// TIA Portal V16 export
// export: Created 2021-04-06T19:52:16.9011384Z, ExportSetting WithDefaults, DisplayName Totally Integrated Automation Portal, DisplayVersion V16, DisplayName TIA Portal Version Control Interface, DisplayVersion V16, DisplayName TIA Portal Openness, DisplayVersion V16, DisplayName STEP 7 Professional, DisplayVersion V16, DisplayName STEP 7 Safety, DisplayVersion V16, DisplayName WinCC Unified SCADA Engineering System, DisplayVersion V16
FUNCTION_BLOCK "workInConveyer_AM"   // FB6, LAD
{ S7_Optimized_Access := 'TRUE' }
VERSION : 0.1
// stored: AutoNumber true, IsIECCheckEnabled false, IsRetainMemResEnabled false, MemoryReserve 100, SetENOAutomatically false, UDAEnableTagReadback false
   VAR_INPUT
      enableWork : Bool;   // разрешение работы
      "setSpeed%Int" : Int;   // уставка скорости
      sensorOverflow : Bool;   // датчик пересыпа
   END_VAR
   VAR_OUTPUT
      startinConveyor : Bool;   // запуск конвейера
      "setSpeed%Real" : Real;
   END_VAR
   VAR
      tonOverflowTable : TON_TIME;   // задержка на включение сигнала пересыпа
      tofOverflowTable : TOF_TIME;   // задержка на выключение сигнала пересыпа
      isOverFlowTable : Bool;   // сигнал сработки сигнала пересыпа
   END_VAR
BEGIN

REGION Network 1: сигнал сработки сигнала пересыпа
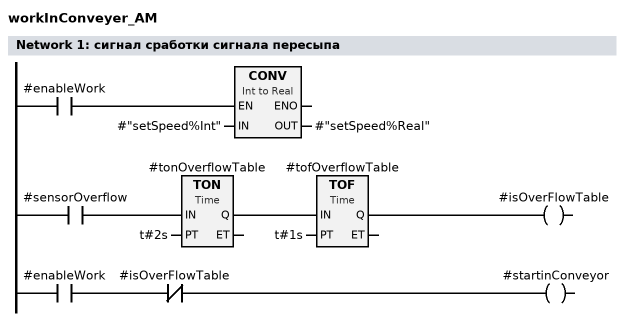
   RUNG wire#powerrail
      Contact( #enableWork )
      { S7_Templates := "[SrcType := Int, DestType := Real]" } Convert(in := #"setSpeed%Int", out => #"setSpeed%Real")
   END_RUNG
   RUNG wire#powerrail
      Contact( #sensorOverflow )
      { S7_Templates := "time_type := Time" } #tonOverflowTable.TON(pt := t#2s, et =>)
      { S7_Templates := "time_type := Time" } #tofOverflowTable.TOF(pt := t#1s, et =>)
      Coil( #isOverFlowTable )
   END_RUNG
   RUNG wire#powerrail
      Contact( #enableWork )
      I_Contact( #isOverFlowTable )
      Coil( #startinConveyor )
   END_RUNG
   // the same network as SCL:
   IF #enableWork THEN #"setSpeed%Real" := INT_TO_REAL(#"setSpeed%Int"); END_IF;
   #tonOverflowTable(IN := #sensorOverflow, PT := t#2s);   // TON
   #tofOverflowTable(IN := #tonOverflowTable.Q, PT := t#1s);   // TOF
   #isOverFlowTable := #tofOverflowTable.Q;
   #startinConveyor := #enableWork AND NOT #isOverFlowTable;
END_REGION
END_FUNCTION_BLOCK
